PROGRAM prgHMIstations
VAR
		tAllStations: BOOL;
	tUsestaions: BOOL;
	btnselectalltrig: R_TRIG;
	btnselall: F_TRIG;
	btnselS1: R_TRIG;
	btnselS2: R_TRIG;
	btnselS3: R_TRIG;
	btnselS4: R_TRIG;
	btnselS5: R_TRIG;
	btnselS6: R_TRIG;

	tPulseStationSelect: BOOL;
	timDelayPulseSelect: TON;
	timPulseStationSelect:TP;
	
END_VAR

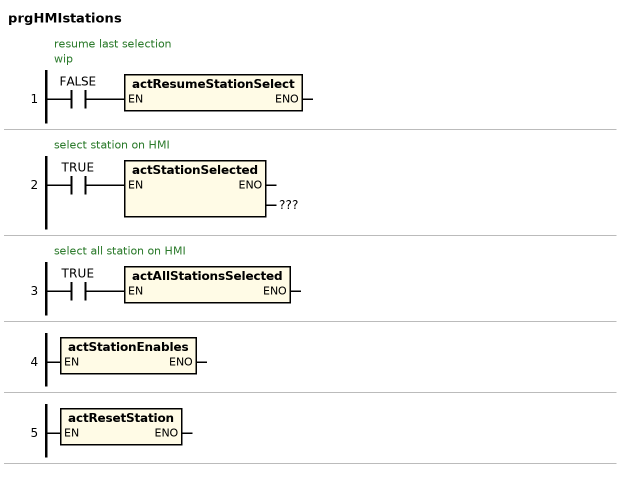
// NETWORK 1
// resume last selection
// wip
IF FALSE THEN actResumeStationSelect(); END_IF

// NETWORK 2
// select station on HMI
actStationSelected();

// NETWORK 3
// select all station on HMI
actAllStationsSelected();

// NETWORK 4
actStationEnables();

// NETWORK 5
actResetStation();

ACTION actAllStationsSelected:
//all station feedback
IF	gHMIData.gStationSelected[1]	AND	
	gHMIData.gStationSelected[2]	AND 
	gHMIData.gStationSelected[3]	AND
	gHMIData.gStationSelected[4]	AND
	gHMIData.gStationSelected[5]	AND
	gHMIData.gStationSelected[6]	
	THEN
		gHMIButtons.btnAllStationsSelected := TRUE;
	ELSE
		gHMIButtons.btnAllStationsSelected := FALSE;
END_IF

//select all stations
btnselectalltrig(CLK:= gHMIButtons.btnSelectAll);
IF btnselectalltrig.Q AND NOT gHMIButtons.btnAllStationsSelected THEN
	gHMIData.gStationSelected[1] := TRUE;
	gHMIData.gStationSelected[2] := TRUE;
	gHMIData.gStationSelected[3] := TRUE;
	gHMIData.gStationSelected[4] := TRUE;
	gHMIData.gStationSelected[5] := TRUE;
	gHMIData.gStationSelected[6] := TRUE;	
END_IF
END_ACTION

ACTION actResetStation:
//if no station is selected, then select station 1
//all station feedback
IF	NOT gHMIData.gStationSelected[1]	AND	
	NOT gHMIData.gStationSelected[2]	AND 
	NOT gHMIData.gStationSelected[3]	AND
	NOT gHMIData.gStationSelected[4]	AND
	NOT gHMIData.gStationSelected[5]	AND
	NOT gHMIData.gStationSelected[6]	
	THEN
		tPulseStationSelect := TRUE;
	ELSE
		tPulseStationSelect := FALSE;
END_IF

//timer delay
timDelayPulseSelect(IN:= tPulseStationSelect, PT:=T#10S);
timPulseStationSelect(IN:=timDelayPulseSelect.Q, PT:=T#1S);

IF timPulseStationSelect.Q THEN
	gHMIData.gActiveStationNumber := 1;
	gHMIData.gStationSelected[1] := TRUE;
END_IF
END_ACTION

ACTION actResumeStationSelect:
//all station feedback
//on select all button falling
btnselall(CLK:= gHMIButtons.btnSelectAll);
IF 	btnselall.Q 					AND
	gHMIData.gStationSelected[1]	AND 
	gHMIData.gStationSelected[2]	AND 
	gHMIData.gStationSelected[3]	AND 
	gHMIData.gStationSelected[4]	AND 
	gHMIData.gStationSelected[5]	AND 
	gHMIData.gStationSelected[6]	 
	THEN

	//clear out selected	
	IF gHMIData.gActiveStationNumber > 1 THEN
		gHMIData.gStationSelected[1] := FALSE;
		gHMIData.gStationSelected[2] := FALSE;
		gHMIData.gStationSelected[3] := FALSE;
		gHMIData.gStationSelected[4] := FALSE;
		gHMIData.gStationSelected[5] := FALSE;
		gHMIData.gStationSelected[6] := FALSE;
	END_IF
	
	//select correct station
	CASE gHMIData.gActiveStationNumber OF
		1:
		gHMIData.gStationSelected[1] := TRUE;
		2:
		gHMIData.gStationSelected[2] := TRUE;
		3:
		gHMIData.gStationSelected[3] := TRUE;
		4:
		gHMIData.gStationSelected[4] := TRUE;
		5:
		gHMIData.gStationSelected[5] := TRUE;
		6:
		gHMIData.gStationSelected[6] := TRUE;
	END_CASE
END_IF
END_ACTION

ACTION actStationEnables:
//disable all stations and let station calls enable on a per-scan basis
gHMIData.gStationEnabled[1]:= System.gSetup.stationEnable[1];
gHMIData.gStationEnabled[2]:= System.gSetup.stationEnable[2];
gHMIData.gStationEnabled[3]:= System.gSetup.stationEnable[3];
gHMIData.gStationEnabled[4]:= System.gSetup.stationEnable[4];
gHMIData.gStationEnabled[5]:= System.gSetup.stationEnable[5];
gHMIData.gStationEnabled[6]:= System.gSetup.stationEnable[6];
END_ACTION

ACTION actStationSelected:
//select station on HMI
//theme:czWR1tA8oB0

btnselS1(clk:=gHMIButtons.btnSelectStation1);
btnselS2(clk:=gHMIButtons.btnSelectStation2);
btnselS3(clk:=gHMIButtons.btnSelectStation3);
btnselS4(clk:=gHMIButtons.btnSelectStation4);
btnselS5(clk:=gHMIButtons.btnSelectStation5);
btnselS6(clk:=gHMIButtons.btnSelectStation6);


//if any button pressed, clear down station memory and prepare for new station selected data
IF	btnselS1.Q OR
	btnselS2.Q OR
	btnselS3.Q OR
	btnselS4.Q OR
	btnselS5.Q OR
	btnselS6.Q
	THEN
		MEMSET(	destAddr:= ADR(gHMIData.gStationSelected),
				fillByte:= 16#0,
				n		:= SIZEOF(gHMIData.gStationSelected)
				);
		gHMIData.gActivePageNumber := 1;
END_IF

//move in correct data next in scan
IF btnselS1.Q THEN
	gHMIData.gActiveStationNumber := 1;
	gHMIData.gStationSelected[1] := TRUE;
END_IF

IF btnselS2.Q THEN
	gHMIData.gActiveStationNumber := 2;
	gHMIData.gStationSelected[2] := TRUE;
END_IF

IF btnselS3.Q THEN
	gHMIData.gActiveStationNumber := 3;
	gHMIData.gStationSelected[3] := TRUE;
END_IF

IF btnselS4.Q THEN
	gHMIData.gActiveStationNumber := 4;
	gHMIData.gStationSelected[4] := TRUE;
END_IF

IF btnselS5.Q THEN
	gHMIData.gActiveStationNumber := 5;
	gHMIData.gStationSelected[5] := TRUE;
END_IF

IF btnselS6.Q THEN
	gHMIData.gActiveStationNumber := 6;
	gHMIData.gStationSelected[6] := TRUE;
END_IF
END_ACTION

END_PROGRAM

(* stored: Version 1.1.0.1, ProductVersion 3.1.4024.11
   POU prgHMIstations: Id {544d1eda-e916-4526-a80c-c42c36049926}, SpecialFunc None
   Action actAllStationsSelected: Id {fc9cc28c-94de-4892-8b94-333e8721262f}
   Action actResetStation: Id {8977bf37-6e2d-0780-3b60-dca3c3d755a0}
   Action actResumeStationSelect: Id {addf1aca-2153-49c7-a870-c5b6bbbacd8b}
   Action actStationEnables: Id {401c3089-158a-4e3f-ba0a-795f1a2a44bf}
   Action actStationSelected: Id {d08ce5bd-f825-4aad-9abb-495ce6676e1e} *)
